FUNCTION_BLOCK SimpleStringBuilder
VAR_INPUT
END_VAR
VAR_OUTPUT
END_VAR
VAR
    builderString: MaxString;
END_VAR

METHOD append
VAR_INPUT
    toAppend: ANY;
END_VAR
VAR
    strToAppend: MaxString;
END_VAR
strToAppend := anyToString(toAppend);
builderString := CONCAT(builderString, strToAppend);
END_METHOD

METHOD toString : MaxString
toString := builderString;
END_METHOD

END_FUNCTION_BLOCK

(* stored: Version 1.1.0.1, ProductVersion 3.1.4022.12
   POU SimpleStringBuilder: Id {cc99bb83-4475-4381-a1e6-019c3040615d}, SpecialFunc None
   Method append: Id {10d89456-de3c-4857-aa02-74792456d045}
   Method toString: Id {b2564f72-8c64-4416-a1f7-a47045c1cdb0} *)
